Staubli VAL3: Motion.pjx

--- Motion.pjx ---
Parameters version=s7.6.2 stackSize=5000 millimeterUnit=true
Program file=checkTrackArea.pgx
Program file=create.pgx
Program file=disableQueue.pgx
Program file=enableQueue.pgx
Program file=flushQueue.pgx
Program file=getConvFrame.pgx
Program file=getConvSpeed.pgx
Program file=getDetectDist.pgx
Program file=getDetectFrame.pgx
Program file=getDistance.pgx
Program file=getErrorMessage.pgx
Program file=getNextID.pgx
Program file=getObjectData.pgx
Program file=getObjectLatch.pgx
Program file=getObjectOffset.pgx
Program file=getRobotArea.pgx
Program file=getStatus.pgx
Program file=getTrackStatus.pgx
Program file=getVersion.pgx
Program file=init.pgx
Program file=kill.pgx
Program file=moveC.pgx
Program file=moveL.pgx
Program file=releaseObject.pgx
Program file=removePart.pgx
Program file=reset.pgx
Program file=resetSignal.pgx
Program file=sendToNextRobot.pgx
Program file=setCalibrating.pgx
Program file=setConvSpeed.pgx
Program file=setConveyor.pgx
Program file=setSignal.pgx
Program file=start.pgx
Program file=stop.pgx
Program file=teach.pgx
Program file=trackOff.pgx
Program file=trackOffJ.pgx
Program file=trackOn.pgx
Program file=trackOnJ.pgx
Program file=trackStopMove.pgx
Program file=tracking.pgx
Program file=whichObjectUsed.pgx
Data file=Motion.dtx
Library alias=cfg path=Disk://Tracking/config/config.pjx autoload=true password=
Library alias=cnv0 path=Disk://Tracking/Templates/GenericConv/GenericConv.pjx autoload=true password=
Library alias=cnv1 path=Disk://Tracking/Templates/GenericConv/GenericConv.pjx autoload=true password=
Library alias=ut path=Disk://Tracking/Tools/util/util.pjx autoload=true password=
Library alias=out path=Disk://Tracking/io/outputs/outputs.pjx autoload=true password=
Library alias=lang path=Disk://Tracking/language/english/english.pjx autoload=true password=

--- Motion.dtx ---
bool bIsScara = true
bool bLinear = true
bool bLizOK = true
bool bReset
bool bSkipVersionChk
bool bStopAll
bool bThruDwnEnabled
bool bThruUpEnabled
dio doThruDwnLimit
dio doThruUpLimit
frame fConveyor = {x=650.958732, y=458.882506, z=-86.396059, rx=0.033285, ry=0.199699, rz=-179.551413, fatherId=world[0]}
frame fMobileFrame[10]
  [0] = {x=3129.225307, fatherId=fConveyor[0]}
  [1] = {x=3129.220405, fatherId=fConveyor[0]}
  [2] = {x=3129.171164, fatherId=fConveyor[0]}
  [3] = {fatherId=fConveyor[0]}
  [4] = {fatherId=fConveyor[0]}
  [5] = {fatherId=fConveyor[0]}
  [6] = {fatherId=fConveyor[0]}
  [7] = {fatherId=fConveyor[0]}
  [8] = {fatherId=fConveyor[0]}
  [9] = {fatherId=fConveyor[0]}
mdesc mTrackOff = {accel=25, vel=50, decel=25, blend=cartesian, leave=20, reach=20}
mdesc mTrackOn = {accel=169, vel=130, decel=169, blend=cartesian, leave=20, reach=20}
mdesc mTracking
num nCnvSynch
num nConveyorSpeed = 518.670703
num nDEFAULTTRKZONE = -99
num nIdxID
num nIdxStatus
num nLinkedTo[10]
  [3] = -1
  [4] = -1
  [5] = -1
  [6] = -1
  [7] = -1
  [8] = -1
  [9] = -1
num nMAXMOBILEFRAME = 10
num nMobFrameSync = -1
num nPosInQueue[10]
  [0] = 2
  [1] = 2
  [2] = 2
  [3] = -1
  [4] = -1
  [5] = -1
  [6] = -1
  [7] = -1
  [8] = -1
  [9] = -1
num nStatus
num nTrackZonPrev = -99
num nTrackingZone = -99
pointRs pInterTrack_RS = {fatherId=fMobileFrame[0]}
pointRs pTrackOff_RS = {x=-127.749433, y=517.878584, z=103.849179, rx=-179.965152, ry=-0.199433, rz=0.448706, shoulder=lefty, fatherId=fConveyor[0]}
pointRs pTrackOn_RS = {x=72.083546, y=72.428021, z=77.085378, rx=-0.209053, ry=-179.916469, rz=-18.008681, shoulder=righty, fatherId=fMobileFrame[2]}
pointRs pTracking_RS = {fatherId=fMobileFrame[0]}
pointRx pInterTrack = {fatherId=fMobileFrame[0]}
pointRx pTrackOff = {fatherId=fConveyor[0]}
pointRx pTrackOn = {fatherId=fMobileFrame[0]}
pointRx pTracking = {fatherId=fMobileFrame[0]}
string sConveyorList = "cvIn"
string sErrMsgList[20]
  [0] = "Not initialized"
  [1] = "Running. No tracking move command pending."
  [2] = "Internal run-time error in task called *\../*. Error code is *. Refer to valTrack Reference guide for more details"
  [3] = "The tracking is in error"
  [4] = "A trackOn command is being executed."
  [5] = "A tracking move command (linear or circular) is being executed."
  [6] = "The arm is tracking a fixed point on a conveyor."
  [9] = "Warning, the add on called "expansion" is required with this VAL3 version"
  [11] = "Warning, libraries for conveyor tracking require VAL3 version s7.6.0 or higher"
  [12] = "MOT>>Number of conveyor is limited to *"
  [13] = "MOT>>The library *\../* used as conveyor number * was not loaded because of error code *"
  [14] = "MOT(init)>>Cannot convert frame number * to mobile frame"
string sErrorMessage = "Running. No tracking move command pending."
string sTASK = "tracking"
tool tTool = {x=-8.16, y=18.26, z=80, rz=110, fatherId=flange[0], ioLink=valve1}

--- getDetectFrame.pgx ---
public program getDetectFrame(num x_nConvNum (dimensions=1), frame& x_fDetectFrame (dimensions=1), frame x_fRefFrame (dimensions=1), num& x_nError (dimensions=1))
begin
  // This program returns the position and orientation of the detection
  //  device frame in reference to the frame x_fRefFrame.
  //
  // Input Param
  //  x_nConvNum : Conveyor number
  //  x_fRefFrame: Reference frame from which the coordinates of
  //                x_fDetection should be returned.
  //
  // Output param
  //  x_fDetection: Coordinates of the detection device frame that have
  //                 been taught during calibration.
  //  x_nError    : Error code
  //    0    --> No error
  //    14   --> Conveyor library not started, the frame cannot be computed.
  //
  //----------------------------------------------------------------
  //
  switch x_nConvNum
    case 0
      if cnv0:libExist("getDetectFrame()")
        call cnv0:getDetectFrame(x_fDetectFrame,x_fRefFrame,x_nError)
      else
        nStatus=-1
      endIf
    break
    case 1
      if cnv1:libExist("getDetectFrame()")
        call cnv1:getDetectFrame(x_fDetectFrame,x_fRefFrame,x_nError)
      else
        nStatus=-1
      endIf
    break
  endSwitch
end

--- getDistance.pgx ---
public program getDistance(num x_nConvNum (dimensions=1), point x_pLoc (dimensions=1), num x_nTime (dimensions=1), num& x_nDist2Up[] (dimensions=1), num& x_nDist2Down[] (dimensions=1), num& x_nError[] (dimensions=1))
begin
  // This program returns the distance between the first object in the
  //  queue and the upstream/downstream limit of the working window.
  //  A negative value means that the object has not reached the
  //  considered limit of the working window. Once the object has
  //  passed the considered limit of the working window, the value of
  //  the returned parameters x_nDist2Up/ x_nDist2Down is positive.
  //
  // Input Param
  //  x_nConvNum      : Conveyor number
  //  x_pLoc          : Original position of the first object in the
  //                     queue. It is the position given by the
  //                     detection device or the position taught with
  //                     the teach() program.
  //  x_nTime         : Time to look ahead to evaluate position of the
  //                     object.
  //
  // Output param
  //  x_fDetection    : Coordinates of the detection device frame that
  //                     have been taught during calibration.
  //  x_nDist2Up      : Distance between location pLoc passed as
  //                     parameter and the upstream limit of the
  //                     working window. The value is positive if the
  //                     object is downstream of the upstream limit
  //                     of the working window.
  //  x_nDist2Down    : Distance between location pLoc passed as
  //                     parameter and downstream end of the working
  //                     window. The value is positive if the object
  //                     is downstream of the downstream limit of the
  //                     working window.
  //  x_nError        :	Error code.
  //                0 = No error
  //                1 = No object with "read" status. This happens
  //                     when program getNextID() has not been
  //                     called.
  //                2 = The object with current ID is not calibrated.
  //                     The teach()program has not been performed
  //                     for this object ID.
  //
  //----------------------------------------------------------------
  //
  switch x_nConvNum
    case 0
      call cnv0:getDistance(x_pLoc,x_nTime,x_nDist2Up,x_nDist2Down,x_nError)
    break
    case 1
      call cnv1:getDistance(x_pLoc,x_nTime,x_nDist2Up,x_nDist2Down,x_nError)
    break
  endSwitch
end

--- getRobotArea.pgx ---
public program getRobotArea(num x_nConvNum (dimensions=1), num& x_nAreaNumber[] (dimensions=1))
begin
  // This program returns in which area number is currently located
  //
  // Input Param
  // x_nConvNum    : Conveyor number
  //
  // Output param
  // x_nAreNumber  : Number of the area in hich is the robot
  //           --> -1: Invalid parameter
  //           --> 0 : robot is beside or above the conveyor
  //           --> 1 : Robot is upstream of the upstream end of the tracking window
  //           --> 2 : Robot is within tracking window
  //           --> 3 : Robot is downstream of the downstream end of the tracking window
  //
  //----------------------------------------------------------------
  //
  if (x_nConvNum>0) and (x_nConvNum<=size(nTrackingZone)-1)
    x_nAreaNumber=nTrackingZone[x_nConvNum]
  else
    x_nAreaNumber=-1
  endIf
end

--- getVersion.pgx ---
public program getVersion(string& x_sVersion[] (dimensions=1))
begin
  // This program returns the version number of the library
  //
  // Input Param
  //  none       :
  //
  // Output param
  //  x_sVersion  : Software version
  //
  //----------------------------------------------------------------
  //
  x_sVersion=cfg:sVERSION
end

--- kill.pgx ---
public program kill()
  local bool l_bMobFrInUse
  local num l_i
begin
  // This program stops all tracking tasks.
  //
  // Input Param
  //  none       :
  //
  // Output param
  //  none       :
  //
  //----------------------------------------------------------------
  //
  // Wait until all tracking movements are finished
  do
    l_bMobFrInUse=false
    for l_i=0 to size(fMobileFrame)-1
      l_bMobFrInUse=(!$setMobile(fMobileFrame[l_i],false) or l_bMobFrInUse)
    endFor
  until l_bMobFrInUse==false
  //
  // Stop task(s) created in this library
  bStopAll=true
  //
  // Request to stop all task of the conveyor libraries
  for l_i=0 to size(sConveyorList)-1
    switch l_i
      case 0
        call cnv0:kill(0)
        // Make sure tasks have been stopped
        watch((taskStatus(sTASK[0]+toString("",0))!=1),2)
      break
      case 1
        call cnv1:kill(1)
        // Make sure tasks have been stopped
        watch((taskStatus(sTASK[0]+toString("",1))!=1),2)
      break
    endSwitch
  endFor
end
